Staubli VAL3: toJointArrayRad.pgx

public program toJointArrayRad(joint& x_jJoint, num& x_nJointArray[])
  local num l_nDeg2Rad
  local num l_nMm2M
begin
  // Copyright (c) 2016, Ocado Technology - Robotics Research Team
  //
  // Licensed under the Apache License, Version 2.0 (the "License");
  // you may not use this file except in compliance with the License.
  // You may obtain a copy of the License at
  //
  //     http://www.apache.org/licenses/LICENSE-2.0
  //
  // Unless required by applicable law or agreed to in writing, software
  // distributed under the License is distributed on an "AS IS" BASIS,
  // WITHOUT WARRANTIES OR CONDITIONS OF ANY KIND, either express or implied.
  // See the License for the specific language governing permissions and
  // limitations under the License.



  l_nDeg2Rad = 0.01745329251
  l_nMm2M = 0.001

  // RS60/RS-TS-safe mapping: first three axes are revolute (deg->rad),
  // fourth axis is linear (mm->m).
  x_nJointArray[0] = x_jJoint.j1 * l_nDeg2Rad
  x_nJointArray[1] = x_jJoint.j2 * l_nDeg2Rad
  x_nJointArray[2] = x_jJoint.j3 * l_nDeg2Rad
  x_nJointArray[3] = x_jJoint.j4 * l_nMm2M
  x_nJointArray[4] = 0
  x_nJointArray[5] = 0
end
